(* PLC project Untitled1.project, CODESYS CODESYS V3.5 SP19 Patch 2 *)
(* stored: creationDateTime 2024-10-03T10:19:48.2662044, modificationDateTime 2024-10-03T10:12:01.335834 *)

PROGRAM PLC_PRG
  VAR
    TEST : BOOL;
  END_VAR

            TEST := TRUE;
          
END_PROGRAM
